PROGRAM OverridePressure
VAR
	fb_SetPressure : FB_SetChamberPressure; 
END_VAR

fb_SetPressure(chamber := stVl_KMono, rNewPressure := New_Pressure, Override:= Global_OverridePressure);

END_PROGRAM

(* stored: Version 1.1.0.1, ProductVersion 3.1.4020.12
   POU OverridePressure: Id {21cef58f-88d1-4cfa-8ccf-34a478fc7cec}, SpecialFunc None *)
